PROGRAM MAIN
VAR
	fbPower: MC_Power;
	EnableAxis1 : BOOL;
	AxisEnabled : BOOL;
	Error : BOOL;
	ErrorID: UDINT;
	
	fbJog: MC_Jog;	
	JogForwardPB : BOOL;
	JogBackwardPB : BOOL;
	
	
	fbReadStatus: MC_ReadStatus;
	AxisStatus: ST_AxisStatus;
	

	inAccel: BOOL;

	JogError: BOOL;
	JogErrorID: UDINT;
END_VAR

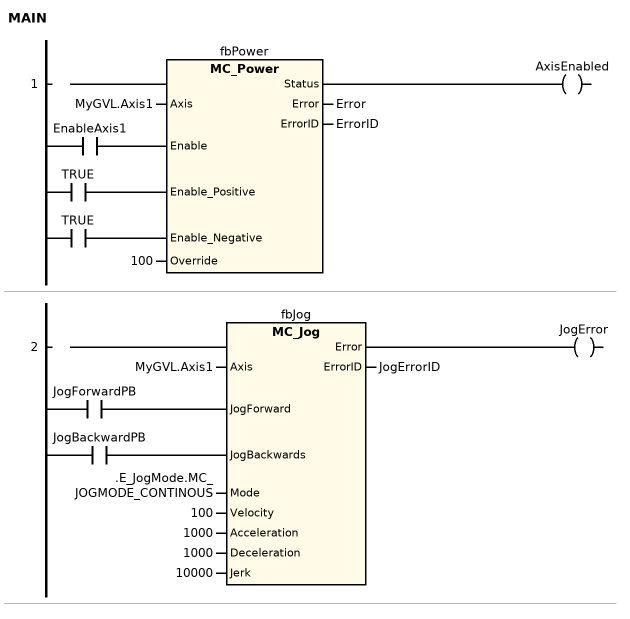
// NETWORK 1
fbPower(
    Axis := MyGVL.Axis1,
    Enable := EnableAxis1,
    Enable_Positive := TRUE,
    Enable_Negative := TRUE,
    Override := 100,
    Error => Error,
    ErrorID => ErrorID); // MC_Power
AxisEnabled := fbPower.Status;

// NETWORK 2
fbJog(
    Axis := MyGVL.Axis1,
    JogForward := JogForwardPB,
    JogBackwards := JogBackwardPB,
    Mode := .E_JogMode.MC_JOGMODE_CONTINOUS,
    Velocity := 100,
    Acceleration := 1000,
    Deceleration := 1000,
    Jerk := 10000,
    Error => JogError,
    ErrorID => JogErrorID); // MC_Jog

END_PROGRAM

(* stored: Version 1.1.0.1, ProductVersion 3.1.4020.12
   POU MAIN: Id {76a13712-a693-42b5-a67a-925c59cea795}, SpecialFunc None *)
